Staubli VAL3: message.pgx

public program message(string& message[], num index)
// Deutsche IF message
begin
  // lenght of message
  //
  switch index
    case 0
      message="Wollen Sie das folgende Tool benutzen:"
    break
    case 1
      message="< IF ASSISTENT >"
    break
    case 2
      message="Wählen Sie den Typ der zu prüfenden Bedingung"
    break
    case 3
      message="Eingang auswählen"
    break
    case 4
      message="Ausgang auswählen"
    break
    case 5
      message="EMAP-Eingang auswählen"
    break
    case 6
      message="Wählen Sie wie der Befehl ausgeführt wird"
    break
    case 7
      message="Wählen Sie den verknüpften Befehl :"
    break
    case 8
      message="Wählen Sie aus der Liste den: "
    break
  endSwitch
end
